(* CODESYS project twoWaterTanksFuncAndBlockContinued.export

Project tree, tasks and I/O mapping:
  Device : CODESYS Control Win V3 x64, CODESYS, version 3.5.22.30
    application Application
      libraries: Standard, 3.5.22.0 (System)
      task MainTask (cyclic, interval t#20ms, priority 1) calls PLC_PRG
      function block FB_Tank [LD]
      function FC_Timer [LD]
      program PLC_PRG [LD]
      Symbols
*)

// Device/Application/PLC_PRG
PROGRAM PLC_PRG
VAR
	FB_Tank_1: FB_Tank;
	Fill: BOOL;
	Discharge: BOOL;
	Fill_Valve: BOOL;
	Fill_ET: TIME;
	Discharge_ET: TIME;
	Discharge_Valve: BOOL;
	Timer: INT;
	FB_Tank_2: FB_Tank;
	Fill2: BOOL;
	Discharge2: BOOL;
	Fill_Valve2: BOOL;
	Fill_ET2: TIME;
	Discharge_ET2: TIME;
	Discharge_Valve2: BOOL;
	Timer2: INT;
END_VAR

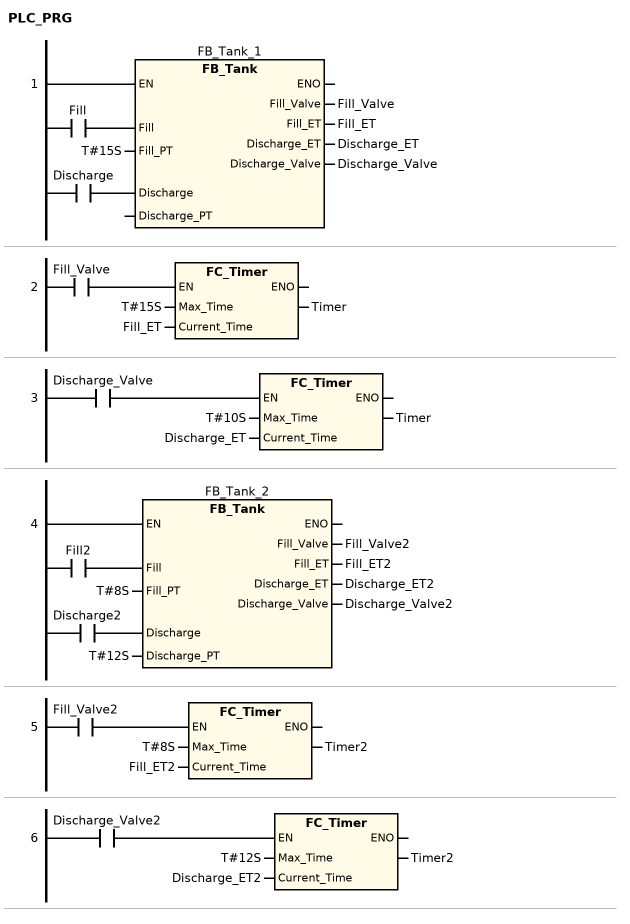
// NETWORK 1
FB_Tank_1(
    Fill := Fill,
    Fill_PT := T#15S,
    Discharge := Discharge,
    Fill_Valve => Fill_Valve,
    Fill_ET => Fill_ET,
    Discharge_ET => Discharge_ET,
    Discharge_Valve => Discharge_Valve); // FB_Tank

// NETWORK 2
IF Fill_Valve THEN Timer := FC_Timer(Max_Time := T#15S, Current_Time := Fill_ET); END_IF

// NETWORK 3
IF Discharge_Valve THEN Timer := FC_Timer(Max_Time := T#10S, Current_Time := Discharge_ET); END_IF

// NETWORK 4
FB_Tank_2(
    Fill := Fill2,
    Fill_PT := T#8S,
    Discharge := Discharge2,
    Discharge_PT := T#12S,
    Fill_Valve => Fill_Valve2,
    Fill_ET => Fill_ET2,
    Discharge_ET => Discharge_ET2,
    Discharge_Valve => Discharge_Valve2); // FB_Tank

// NETWORK 5
IF Fill_Valve2 THEN Timer2 := FC_Timer(Max_Time := T#8S, Current_Time := Fill_ET2); END_IF

// NETWORK 6
IF Discharge_Valve2 THEN Timer2 := FC_Timer(Max_Time := T#12S, Current_Time := Discharge_ET2); END_IF

END_PROGRAM

// Device/Application/FB_Tank
FUNCTION_BLOCK FB_Tank
VAR_INPUT
	Fill: BOOL;
	Fill_PT: TIME := T#10S;
	Discharge: BOOL;
	Discharge_PT: TIME := T#10s;
END_VAR
VAR_OUTPUT
	Fill_Valve: BOOL;
	Fill_ET: TIME;
	Discharge_ET: TIME;
	Discharge_Valve: BOOL;
END_VAR
VAR
	TP_0: TP;

	TP_1: TP;
END_VAR
VAR // added by the converter: edge detectors and wires of the graphical bodies
    _rt1 : R_TRIG;
    _ft1 : F_TRIG;
END_VAR

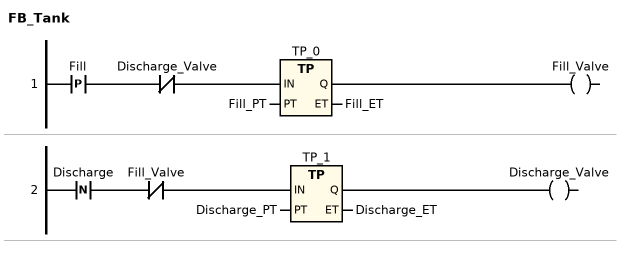
// NETWORK 1
_rt1(CLK := Fill);
TP_0(IN := _rt1.Q AND NOT Discharge_Valve, PT := Fill_PT, ET => Fill_ET); // TP
Fill_Valve := TP_0.Q;

// NETWORK 2
_ft1(CLK := Discharge);
TP_1(IN := _ft1.Q AND NOT Fill_Valve, PT := Discharge_PT, ET => Discharge_ET); // TP
Discharge_Valve := TP_1.Q;

END_FUNCTION_BLOCK

// Device/Application/FC_Timer
FUNCTION FC_Timer : INT
VAR_INPUT
	Max_Time: TIME;
	Current_Time: TIME;
END_VAR
VAR

	Var1: TIME;
	Inv_Time_INT: INT;
END_VAR

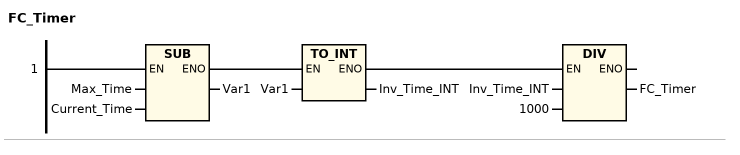
// NETWORK 1
Var1 := Max_Time - Current_Time;
Inv_Time_INT := TO_INT(Var1);
FC_Timer := Inv_Time_INT / 1000;

END_FUNCTION
